PROGRAM MAIN
VAR
	
END_VAR

SignalmappingInput();
Call_HMI();
Call_Emitter();
Call_OperatingMode();
// Call_Foerderband();
Call_Aufzug();
Call_Warehouse();
Call_RFID();
Call_VisionSensor();
SignalmappingOutput();

END_PROGRAM

(* stored: Version 1.1.0.1
   POU MAIN: Id {7aa52cb8-d531-4a9c-a3e7-eb662cc7341b}, SpecialFunc None *)
